Yaskawa INFORM job: R2_W70(-90,-90)AWMOZEOK.JBI

/JOB
//NAME R2_W70(-90,-90)AWMOZEOK
///FOLDERNAME AWOK
//POS
///NPOS 46,46,0,2,0,0
///TOOL 0
///POSTYPE PULSE
///PULSE
C00000=102427,12534,-18173,-7407,79911,17289
C00001=160789,-105634,-92335,-27114,52891,-64558
C00002=121171,-45685,-64164,-545,59125,-81793
C00003=121163,-42376,-62156,-538,59589,-81798
C00004=121160,-41064,-61345,-535,59765,-81800
C00005=121171,-45049,-63783,-545,59217,-81793
C00006=121166,-43227,-62678,-541,59473,-81796
C00007=121171,-45049,-63783,-545,59217,-81793
C00008=121160,-41064,-61345,-535,59765,-81800
C00009=121150,-37084,-58834,-526,60264,-81806
C00010=121154,-38695,-59859,-530,60067,-81804
C00011=121150,-37084,-58834,-526,60264,-81806
C00012=121160,-41064,-61345,-535,59765,-81800
C00013=121157,-40054,-60715,-533,59896,-81802
C00014=121152,-37732,-59248,-528,60186,-81805
C00015=121152,-37737,-59251,-528,60185,-81805
C00016=121152,-37732,-59248,-528,60186,-81805
C00017=121157,-40054,-60715,-533,59896,-81802
C00018=121160,-41064,-61345,-535,59765,-81800
C00019=121163,-42376,-62156,-538,59589,-81798
C00020=121171,-45685,-64164,-545,59125,-81793
C00021=86344,37741,16232,-33234,79198,-22875
C00022=86348,41355,36711,-34748,70202,-20064
C00023=86758,45970,45114,-35406,68058,-19166
C00024=86920,48010,48733,-35704,67157,-18784
C00025=86908,47205,46567,-35491,67906,-19048
C00026=87315,45639,45695,-35622,67855,-18851
C00027=87923,56522,58366,-37180,67863,-17361
C00028=90013,81259,88089,-39267,65144,-14735
C00029=90671,95980,107303,-40951,62963,-12848
C00030=90560,89177,96837,-40047,65183,-13837
C00031=90277,78829,80053,-38736,68980,-15473
C00032=90274,68501,50557,-36666,79273,-19158
C00033=84587,45041,21539,-15707,66208,-49808
C00034=84591,48499,41963,-17363,55841,-48233
C00035=85040,53724,51591,-18270,52847,-47511
C00036=85216,56096,55819,-18688,51572,-47192
C00037=84975,53615,52169,-18337,52441,-47464
C00038=85221,55266,53593,-18460,52470,-47361
C00039=85218,56098,55804,-18690,51593,-47195
C00040=85218,56092,55792,-18688,51597,-47195
C00041=85214,56055,55741,-18680,51597,-47198
C00042=85037,53687,51518,-18263,52871,-47516
C00043=84588,48468,41898,-17358,55863,-48238
C00044=84584,45025,21492,-15704,66228,-49811
C00045=84726,45334,21315,-15735,66513,-49797
BC00000=159258,359476,995204
BC00001=208039,-35650,857774
BC00002=208047,-36082,880468
BC00003=208095,-36082,855898
BC00004=208114,-36082,846070
BC00005=208149,-36082,831548
BC00006=208158,-36082,826145
BC00007=208149,-36082,831548
BC00008=208114,-36082,846070
BC00009=208128,-36082,840660
BC00010=208143,-36082,834673
BC00011=208128,-36082,840660
BC00012=208114,-36082,846070
BC00013=199007,-36082,849498
BC00014=199052,-36082,826827
BC00015=201441,-36082,826884
BC00016=199052,-36082,826827
BC00017=199007,-36082,849498
BC00018=208114,-36082,846070
BC00019=208095,-36082,855898
BC00020=208047,-36082,880468
BC00021=28998,-36082,1075175
BC00022=29039,-36082,1075175
BC00023=32496,-36082,1075175
BC00024=33879,-36082,1075175
BC00025=33879,-36082,1075175
BC00026=33879,-36082,1075175
BC00027=30845,-36082,1075175
BC00028=22638,-36082,1075175
BC00029=20121,-36082,1075175
BC00030=18626,-36082,1075175
BC00031=14891,-36082,1075175
BC00032=14850,-36082,1075175
BC00033=47575,0,1075175
BC00034=47617,0,1075175
BC00035=48359,0,1075175
BC00036=48656,0,1075175
BC00037=48656,0,1075175
BC00038=48656,0,1075175
BC00039=52201,0,1075175
BC00040=53434,0,1075175
BC00041=56979,0,1075175
BC00042=56682,0,1075175
BC00043=55940,0,1075175
BC00044=55898,0,1075175
BC00045=55898,399813,1075175
///POSTYPE BASE
///RECTAN
///RCONF 0,0,0,0,1,0,0,0,0,0,0,0,0,0,0,0,0,0,0,0,0,0,0,0
P00006=2.006,1.622,-0.565,0.0000,0.0000,0.0000
///RCONF 0,0,0,0,0,0,0,0,0,0,0,0,0,0,0,0,0,0,0,0,0,0,0,0
P00023=-2.957,-4.083,2.762,0.0000,0.0000,0.0000
//INST
///DATE 2023/11/16 14:20
///ATTR SC,RW
///GROUP1 RB1,BS1
NOP
'r2_W70(-90,-90)
'Path S807
MOVJ C00000 BC00000 VJ=20.00
SFTOF
MOVJ C00001 BC00001 VJ=20.00
DOUT OG#(200) 10
WAIT IG#(200)=10
MOVJ C00002 BC00002 VJ=20.00
MOVL C00003 BC00003 V=100.0
MOVL C00004 BC00004 V=100.0
MOVL C00005 BC00005 V=60.0
REFP 3 C00006 BC00006
CALL JOB:SEARCH-R1
SET P023 P006
SFTON P023
MOVL C00007 BC00007 V=60.0
MOVL C00008 BC00008 V=100.0
MOVL C00009 BC00009 V=60.0
REFP 3 C00010 BC00010
CALL JOB:SEARCH-R1
SET P023 P006
SFTON P023
MOVL C00011 BC00011 V=60.0
MOVL C00012 BC00012 V=100.0
MOVL C00013 BC00013 V=100.0
MOVL C00014 BC00014 V=60.0
REFP 3 C00015 BC00015
CALL JOB:SEARCH-R1
SET P023 P006
SFTON P023
MOVL C00016 BC00016 V=60.0
MOVL C00017 BC00017 V=100.0
MOVL C00018 BC00018 V=100.0
MOVL C00019 BC00019 V=100.0
MOVL C00020 BC00020 V=100.0
'Path W104
SFTOF
SFTON P023
MOVJ C00021 BC00021 VJ=20.00
MOVJ C00022 BC00022 VJ=20.00
MOVL C00023 BC00023 V=100.0
MOVL C00024 BC00024 V=100.0 PL=0
REFP 1 C00025 BC00025
REFP 2 C00026 BC00026
MACRO1 MJ#(0) ARGF0
COMM ARCON
MOVL C00027 BC00027 V=10.0
MOVL C00028 BC00028 V=10.0
MOVL C00029 BC00029 V=10.0
ARCOF
MOVL C00030 BC00030 V=100.0
MOVL C00031 BC00031 V=100.0
MOVL C00032 BC00032 V=100.0
SFTOF
'Path W103
SFTOF
SFTON P023
MOVJ C00033 BC00033 VJ=20.00
MOVJ C00034 BC00034 VJ=20.00
MOVL C00035 BC00035 V=100.0
MOVL C00036 BC00036 V=100.0 PL=0
REFP 1 C00037 BC00037
REFP 2 C00038 BC00038
MACRO1 MJ#(0) ARGF9
COMM ARCON
MOVL C00039 BC00039 V=10.0
MOVL C00040 BC00040 V=10.0
MOVL C00041 BC00041 V=10.0
ARCOF
MOVL C00042 BC00042 V=100.0
MOVL C00043 BC00043 V=100.0
MOVL C00044 BC00044 V=100.0
SFTOF
MOVJ C00045 BC00045 VJ=20.00
END
